// TIA Portal V19 export
FUNCTION_BLOCK "TYPIC_C701_IF_KLB"   // FB120, FBD
TITLE = TYPIC_C701_IF_KLB: Brandklep
{ S7_Optimized_Access := 'TRUE' }
AUTHOR : OCOTECH
FAMILY : Typical
NAME : C701.708
// Logisch Object Besturing: C701.708
// 
// De interne functie Brandklep verzorgt de interne besturing, bewaking en fysieke aansturing van een brandklep.
// stored: MemoryReserve 10, SetENOAutomatically false
   VAR_INPUT
      IN_KLB { ExternalAccessible := 'False'; ExternalVisible := 'False'; ExternalWritable := 'False'} : Bool;   // Status brandklep (1 = Open)
   END_VAR
   VAR_OUTPUT
      VAR_IF_KLB { ExternalAccessible := 'False'; ExternalVisible := 'False'; ExternalWritable := 'False'} : "C701_VAR_IF_KLB_TYPIC";   // Struct met alle variabelen naar bovenliggende functies
   END_VAR
   VAR
      STO { ExternalWritable := 'False'} : Struct   // Storingen
         A001 : Bool;   // Brandklep gesloten
      END_STRUCT;
      VAR { ExternalWritable := 'False'} : Struct   // Variabelen
         KLB_TOE { ExternalAccessible := 'False'; ExternalVisible := 'False'} : Bool;   // Brandklep gesloten
      END_STRUCT;
   END_VAR
BEGIN

REGION Network 1: START
END_REGION

REGION Network 2: +++ Storingen +++
   // aanmaken storingen.
END_REGION

REGION Network 3: Storing A001: Brandklep gesloten
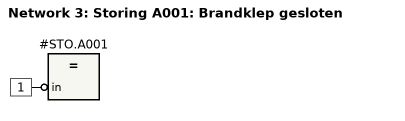
   #STO.A001 := NOT 1;
END_REGION

REGION Network 4 (SCL): EINDE
   // Variabelen van intern scada rakvlak naar outputs copieren
   #VAR_IF_KLB.KLB_TOE := #VAR.KLB_TOE;
END_REGION
END_FUNCTION_BLOCK
